// TwinCAT 3 PLC project EXERCISES
// ProgramVersion: 3.1.4023.0
// libraries:
//   CmpBitmapPool, * (System)
//   Tc2_Standard, * (Beckhoff Automation GmbH)
//   Tc2_System, * (Beckhoff Automation GmbH)
//   Tc2_Utilities, * (Beckhoff Automation GmbH)
//   Tc3_Module, * (Beckhoff Automation GmbH)
// project tree:
//   DUTs/ Pers_Data.TcDUT
//   / GlobalTextList.TcGTLO, ImagePool.TcIPO (not stored), PlcTask.TcTTO, Visualization Manager.TcVMO (not stored)
//   POUs/ Auto_Deur.TcPOU, Belsig_Winkeldeur.TcPOU, Check_Bounds_15_TO_24.TcPOU, FB_PULSE_PER_X_SEC.TcPOU, FB_PWM.TcPOU, Knipperlicht.TcPOU, MAIN.TcPOU, Open_Toilet.TcPOU, Parking.TcPOU, FC_SCALE.TcPOU, Product_Tellen_Verdelen.TcPOU, FB_String_Search.TcPOU, Trappenhuisautomaat.TcPOU
//   VISUs/ Auto_Deur.TcVIS, Belsig_Winkeldeur.TcVIS, Knipperlicht.TcVIS, Open_Toilet.TcVIS, Parking.TcVIS, Product_Tellen_Verdelen.TcVIS, Trappenhuisautomaat.TcVIS
// real-time tasks:
//   TASK PlcTask: cycle T#10ms, priority 20, ADS port 350

CONFIGURATION EXERCISES
    RESOURCE PLC ON TwinCAT3
        TASK PlcTask(INTERVAL := T#10ms, PRIORITY := 20);
        PROGRAM MAIN WITH PlcTask : MAIN;
    END_RESOURCE
END_CONFIGURATION

// ---- DUTs/Pers_Data.TcDUT
TYPE Pers_Data :
STRUCT
	Name : STRING;
	Firstname :  STRING;
	Age : STRING;
	Address : STRING;
END_STRUCT
END_TYPE

// ---- POUs/MAIN.TcPOU
PROGRAM MAIN
VAR
	KASPER : UINT;
	FB_PWM : FB_PWM;
	PWM : BOOL;
END_VAR

FB_PWM(DUTY:= 50, PERIOD_MS:= 4000);

PWM := FB_PWM.PWM_SIGNAL;

END_PROGRAM

// ---- POUs/FB_PWM.TcPOU
FUNCTION_BLOCK FB_PWM

VAR_INPUT
	DUTY : UINT;
	PERIOD_MS : UINT;
END_VAR

VAR_OUTPUT
	PWM_SIGNAL : BOOL;
END_VAR

VAR
	ON_TIME_STR : STRING;
	OFF_TIME_STR : STRING;
	
	ON_TIME : TIME;
	OFF_TIME : TIME;
	
	TON : TON;
	TOF : TOF;
END_VAR

ON_TIME_STR := UINT_TO_STRING(DUTY * PERIOD_MS / 100);
ON_TIME_STR := CONCAT('T#', ON_TIME_STR);
ON_TIME_STR := CONCAT(ON_TIME_STR, 'ms');
ON_TIME := STRING_TO_TIME(ON_TIME_STR);
	
OFF_TIME_STR := UINT_TO_STRING(PERIOD_MS - (DUTY * PERIOD_MS / 100));
OFF_TIME_STR := CONCAT('T#', OFF_TIME_STR);
OFF_TIME_STR := CONCAT(OFF_TIME_STR, 'ms');
OFF_TIME := STRING_TO_TIME(OFF_TIME_STR);

TOF(IN:= TON.Q, PT:= ON_TIME, Q => PWM_SIGNAL);
TON(IN:= NOT(TOF.Q), PT:= OFF_TIME);

END_FUNCTION_BLOCK

// ---- POUs/Auto_Deur.TcPOU
PROGRAM Auto_Deur
VAR
	TOF : TOF;
END_VAR

VAR_INPUT
	SW_MAIN : BOOL;
	SW_KASSA : BOOL;
	SENSOR_DOOR : BOOL;
END_VAR

VAR_OUTPUT
	CIL : BOOL;
END_VAR

IF SW_MAIN THEN
	TOF(IN:= SW_KASSA OR SENSOR_DOOR, PT:= T#1S, Q=> CIL);
END_IF

END_PROGRAM

// ---- POUs/Belsig_Winkeldeur.TcPOU
PROGRAM Belsig_Winkeldeur
VAR
	CTU : CTU;
	R_TRIG : R_TRIG;
	R_TRIG2 : R_TRIG;
END_VAR

VAR_INPUT
	S01 : BOOL;
	S02 : BOOL;
END_VAR

VAR_OUTPUT
	Q00 : BOOL;
END_VAR

CTU(CU := R_TRIG.Q);
R_TRIG(CLK := Q00);
R_TRIG2(CLK := S02);

IF S01 THEN
	IF R_TRIG2.Q THEN
		Q00 := TRUE;
	END_IF
	
ELSIF Q00 THEN
	IF S02 THEN
		Q00 := TRUE;
	ELSE
		Q00 := FALSE;
	END_IF
END_IF

END_PROGRAM

// ---- POUs/Check_Bounds_15_TO_24.TcPOU
FUNCTION Check_Bounds_15_TO_24 : BOOL

VAR_INPUT
	Value : UINT;
END_VAR

IF VALUE <= 24 AND VALUE >= 15 THEN
	Check_Bounds_15_TO_24 := TRUE;
ELSE
	Check_Bounds_15_TO_24 := FALSE;
END_IF

END_FUNCTION

// ---- POUs/FB_PULSE_PER_X_SEC.TcPOU
FUNCTION_BLOCK FB_PULSE_PER_X_SEC
VAR_INPUT
	ON_OFF : BOOL;
	X_Sec : UINT;
END_VAR

VAR_OUTPUT
	PULSE : BOOL;
END_VAR

VAR
	R_TRIG : R_TRIG;
	TIMETIME : TIME;
	TIME_TIJD : STRING;
	TON : TON;
	TOF : TOF;
END_VAR

TIME_TIJD := CONCAT('T#', UINT_TO_STRING(X_Sec));
TIME_TIJD := CONCAT(TIME_TIJD, 's');

TOF(IN:= TON.Q, PT:= T#0MS);
TON(IN:= NOT(TOF.Q), PT:= STRING_TO_TIME(TIME_TIJD), Q => Pulse);

END_FUNCTION_BLOCK

// ---- POUs/Knipperlicht.TcPOU
PROGRAM Knipperlicht
VAR
	TOF : TOF;
	TON : TON;
END_VAR

VAR_OUTPUT
	LAMP : BOOL;
END_VAR

TOF(IN:= TON.Q, PT:= T#500MS, Q => LAMP);
TON(IN:= NOT(TOF.Q), PT:= T#500ms);

END_PROGRAM

// ---- POUs/Open_Toilet.TcPOU
PROGRAM Open_Toilet
VAR
	TOF : TOF;
END_VAR

VAR_INPUT
	SW1 : BOOL; // SWITCH 1
	SW2 : BOOL; // SWITCH 2
	SW3 : BOOL; // SWITCH 3
END_VAR

VAR_OUTPUT
	Q00 : BOOL; // VENTILATOR
	Q01 : BOOL; // LAMP 1
	Q02 : BOOL; // LAMP 2
	Q03 : BOOL; // LAMP 3
END_VAR

TOF(IN:= SW1 OR SW2 OR SW3, PT:= T#5S, Q=> Q00);

END_PROGRAM

// ---- POUs/Parking.TcPOU
PROGRAM Parking
VAR
	R_TRIG_1 : R_TRIG;
	R_TRIG_2 : R_TRIG;
	
	R_TRIG_BINNEN : R_TRIG;
	R_TRIG_BUITEN : R_TRIG;
	
	CTUD : CTUD;	
	
	PING1 : BOOL;
	PING2 : BOOL;
	
	BINNEN : BOOL;
	BUITEN : BOOL;
END_VAR

VAR_INPUT
	SENSOR_1 : BOOL;
	SENSOR_2 : BOOL;
END_VAR

VAR_OUTPUT
	LED_R : BOOL;
	LED_G : BOOL;
	SLAGBOOM : BOOL;
END_VAR

R_TRIG_1(CLK := SENSOR_1);
R_TRIG_2(CLK := SENSOR_2);
R_TRIG_BINNEN(CLK := BINNEN);
R_TRIG_BUITEN(CLK := BUITEN);

CTUD(CU := R_TRIG_BINNEN.Q, CD := R_TRIG_BUITEN.Q);

IF R_TRIG_1.Q THEN
	IF PING2 THEN
		BUITEN := TRUE;
		SLAGBOOM := FALSE;
		PING2 := FALSE;
	ELSE
		PING1 := TRUE;
		SLAGBOOM := TRUE;
	END_IF
ELSE
	BUITEN := FALSE;
END_IF

IF R_TRIG_2.Q THEN
	IF PING1 THEN
		BINNEN := TRUE;
		SLAGBOOM := FALSE;
		PING1 := FALSE;
	ELSE
		PING2 := TRUE;
		SLAGBOOM := TRUE;
	END_IF
ELSE
	BINNEN := FALSE;
END_IF

IF CTUD.CV < 10 THEN
	LED_G := TRUE;
	LED_R := FALSE;
ELSE
	LED_R := TRUE;
	LED_G := FALSE;
END_IF

END_PROGRAM

// ---- POUs/FC_SCALE.TcPOU
FUNCTION FC_SCALE : LREAL

VAR_INPUT
	RawValue : LREAL;
	Rvmin : LREAL;
	Rvmax : LREAL;
	SVmin : LREAL;
	SVmax : LREAL;
END_VAR

FC_SCALE := SVmin + (RawValue / ((Rvmax-Rvmin)/(SVmax-SVmin)));

END_FUNCTION

// ---- POUs/Product_Tellen_Verdelen.TcPOU
PROGRAM Product_Tellen_Verdelen
VAR
	R_TRIG : R_TRIG;
	CTU : CTU;
END_VAR

VAR_INPUT
	SENSOR : BOOL;
	STAND_1 : BOOL;
	STAND_2 : BOOL;
END_VAR

VAR_OUTPUT
END_VAR

R_TRIG(CLK := SENSOR);
CTU(CU:= R_TRIG.Q); 

IF CTU.CV < 10 THEN
	CTU.RESET := FALSE;
	STAND_1 := TRUE;
	STAND_2 := FALSE;
ELSIF CTU.CV < 30 THEN
	STAND_1 := FALSE;
	STAND_2 := TRUE;
ELSE
	CTU.RESET := R_TRIG.Q;
END_IF

END_PROGRAM

// ---- POUs/FB_String_Search.TcPOU
FUNCTION_BLOCK FB_String_Search

VAR_INPUT
	InputString : Pers_Data;
	SearchString : STRING;
END_VAR

VAR_OUTPUT
	OUT : BOOL;
END_VAR

VAR
	SUB_STRING : STRING;
END_VAR

SUB_STRING := CONCAT(SUB_STRING, InputString.Name);
SUB_STRING := CONCAT(SUB_STRING, InputString.Firstname);
SUB_STRING := CONCAT(SUB_STRING, InputString.Age);
SUB_STRING := CONCAT(SUB_STRING, InputString.Address);

OUT := INT_TO_BOOL(FIND(STR1:= F_ToLCase(SUB_String), STR2:= F_ToLCase(SearchString)));

END_FUNCTION_BLOCK

// ---- POUs/Trappenhuisautomaat.TcPOU
PROGRAM Trappenhuisautomaat
VAR
	TOF : TOF;
	CTUD : CTUD;
END_VAR

VAR_INPUT
	SW0 : BOOL;
	SW1 : BOOL;
	SW2 : BOOL;
	SW3 : BOOL;
	SW4 : BOOL;
	SW5 : BOOL;
	SW6 : BOOL;
END_VAR

VAR_OUTPUT
	Q01 : BOOL;
END_VAR

TOF(IN:= SW0, PT:= T#3S, Q=> Q01);
CTUD.RESET := NOT(Q01);


IF SW1 OR SW2 OR SW3 OR SW4 OR SW5 OR SW6 THEN
	SW0 := TRUE; 
	CTUD.CU := SW0;
	IF CTUD.CV = 2 THEN
		TOF.PT := T#0S;
		SW0 := FALSE;
		Q01 := FALSE; 
	END_IF
ELSE
	SW0 := FALSE;
END_IF

END_PROGRAM

// ---- GlobalTextList.TcGTLO
TEXTLIST GlobalTextList
  868 = '%d'
  584 = '%ld'
END_TEXTLIST

// ---- VISUs/Auto_Deur.TcVIS
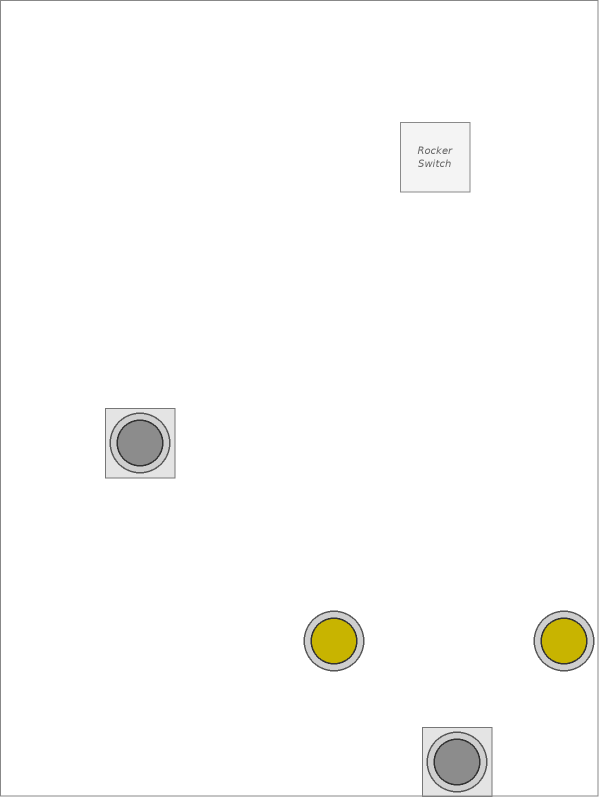
VISUALIZATION Auto_Deur  // 599x797
    Lamp1 (529,606 70x70), variable: Auto_Deur.CIL, style: Lamp-Lamp1-Yellow
    Lamp1 (299,606 70x70), variable: Auto_Deur.CIL, style: Lamp-Lamp1-Yellow
    PushSwitch (422,727 70x70), variable: Auto_Deur.SENSOR_DOOR, behaviour: TAP, style: Switch-PushSwitch-Gray
    PushSwitch (105,408 70x70), variable: Auto_Deur.SW_KASSA, behaviour: TAP, style: Switch-PushSwitch-Gray
    RockerSwitch (400,122 70x70), variable: Auto_Deur.SW_MAIN, behaviour: TOGGLE, style: Switch-RockerSwitch-Gray
END_VISUALIZATION

// ---- VISUs/Belsig_Winkeldeur.TcVIS
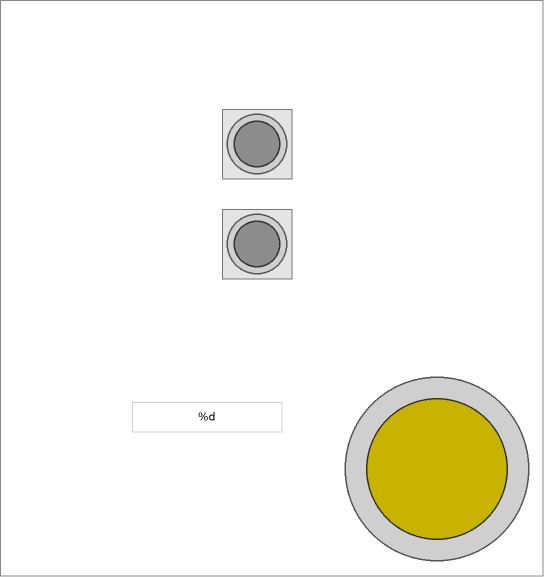
VISUALIZATION Belsig_Winkeldeur  // 544x577
    PushSwitch (222,109 70x70), variable: Belsig_Winkeldeur.S01, behaviour: TOGGLE, style: Switch-PushSwitch-Gray
    PushSwitch (222,209 70x70), variable: Belsig_Winkeldeur.S02, behaviour: TOGGLE, style: Switch-PushSwitch-Gray
    Lamp1 (330,361 214x216), variable: Belsig_Winkeldeur.Q00, style: Lamp-Lamp1-Yellow
    Textfield (132,402 150x30), "%d", text variable: Belsig_Winkeldeur.CTU.CV
END_VISUALIZATION

// ---- VISUs/Knipperlicht.TcVIS
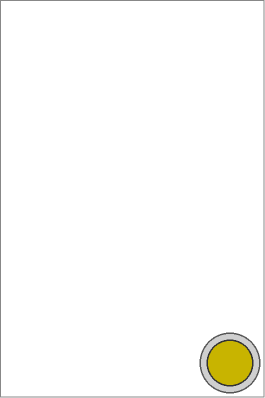
VISUALIZATION Knipperlicht  // 265x398
    Lamp1 (195,328 70x70), variable: Knipperlicht.LAMP, style: Lamp-Lamp1-Yellow
END_VISUALIZATION

// ---- VISUs/Open_Toilet.TcVIS
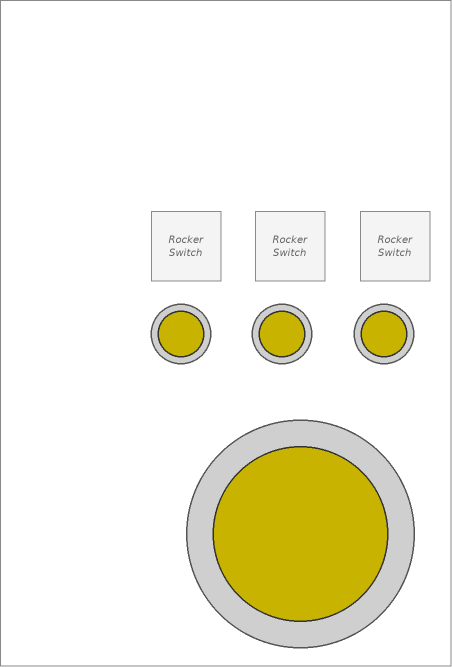
VISUALIZATION Open_Toilet  // 452x667
    Lamp1 (146,299 70x70), variable: Open_Toilet.SW1, style: Lamp-Lamp1-Yellow
    Lamp1 (247,299 70x70), variable: Open_Toilet.SW2, style: Lamp-Lamp1-Yellow
    Lamp1 (349,299 70x70), variable: Open_Toilet.SW3, style: Lamp-Lamp1-Yellow
    Lamp1 (149,401 303x266), variable: Open_Toilet.Q00, style: Lamp-Lamp1-Yellow
    RockerSwitch (151,211 70x70), variable: Open_Toilet.SW1, behaviour: TOGGLE, style: Switch-RockerSwitch-Gray
    RockerSwitch (255,211 70x70), variable: Open_Toilet.SW2, behaviour: TOGGLE, style: Switch-RockerSwitch-Gray
    RockerSwitch (360,211 70x70), variable: Open_Toilet.SW3, behaviour: TOGGLE, style: Switch-RockerSwitch-Gray
END_VISUALIZATION

// ---- VISUs/Parking.TcVIS
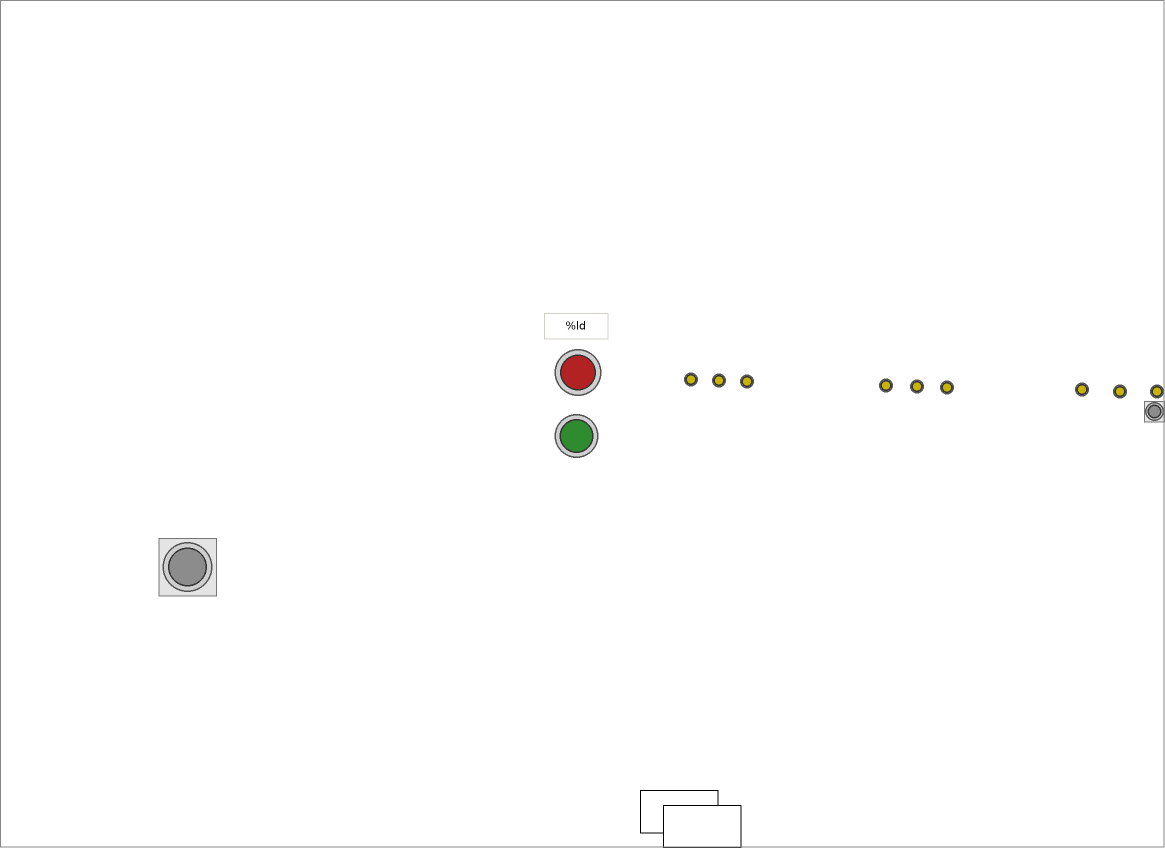
VISUALIZATION Parking  // 1165x848, background image ImagePool.image-3
    Lamp1 (551,345 54x55), variable: Parking.LED_R, style: Lamp-Lamp1-Red
    Lamp1 (551,410 51x52), variable: Parking.LED_G, style: Lamp-Lamp1-Green
    Textfield (544,313 64x26), "%ld", text variable: Parking.CTUD.CV
    PushSwitch (1144,399 21x25), variable: Parking.SENSOR_2, behaviour: TAP, style: Switch-PushSwitch-Gray
    PushSwitch (158,538 59x58), variable: Parking.SENSOR_1, behaviour: TAP, style: Switch-PushSwitch-Gray
    Rectangle (640,790 78x43), angle 69
    Rectangle (663,805 78x43), angle 160
    Lamp1 (683,359 16x41), variable: Parking.SLAGBOOM, style: Lamp-Lamp1-Yellow
    Lamp1 (711,360 16x41), variable: Parking.SLAGBOOM, style: Lamp-Lamp1-Yellow
    Lamp1 (739,361 16x41), variable: Parking.SLAGBOOM, style: Lamp-Lamp1-Yellow
    Lamp1 (878,365 16x41), variable: Parking.SLAGBOOM, style: Lamp-Lamp1-Yellow
    Lamp1 (939,367 16x41), variable: Parking.SLAGBOOM, style: Lamp-Lamp1-Yellow
    Lamp1 (909,366 16x41), variable: Parking.SLAGBOOM, style: Lamp-Lamp1-Yellow
    Lamp1 (1074,369 16x41), variable: Parking.SLAGBOOM, style: Lamp-Lamp1-Yellow
    Lamp1 (1112,370 16x43), variable: Parking.SLAGBOOM, style: Lamp-Lamp1-Yellow
    Lamp1 (1149,371 16x41), variable: Parking.SLAGBOOM, style: Lamp-Lamp1-Yellow
END_VISUALIZATION

// ---- VISUs/Product_Tellen_Verdelen.TcVIS
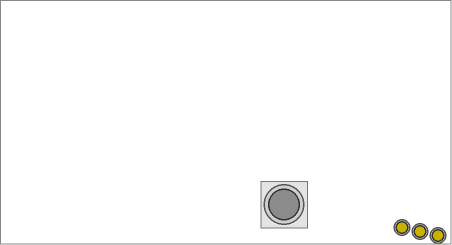
VISUALIZATION Product_Tellen_Verdelen  // 452x245, background image ImagePool.VerdelerFULL
    PushSwitch (259,181 50x47), variable: Product_Tellen_Verdelen.SENSOR, behaviour: TAP, style: Switch-PushSwitch-Gray
    Lamp1 (388,218 28x19), variable: Product_Tellen_Verdelen.STAND_2, style: Lamp-Lamp1-Yellow
    Lamp1 (406,222 28x19), variable: Product_Tellen_Verdelen.STAND_2, style: Lamp-Lamp1-Yellow
    Lamp1 (424,226 28x19), variable: Product_Tellen_Verdelen.STAND_2, style: Lamp-Lamp1-Yellow
END_VISUALIZATION

// ---- VISUs/Trappenhuisautomaat.TcVIS
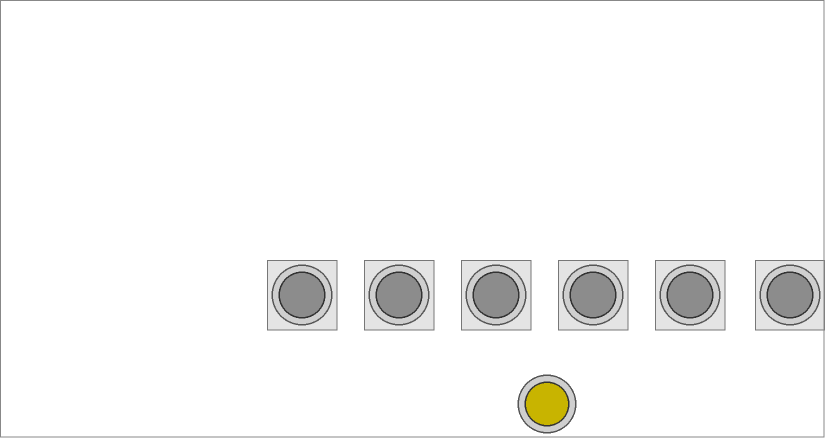
VISUALIZATION Trappenhuisautomaat  // 825x438
    Lamp1 (512,370 70x68), variable: Trappenhuisautomaat.Q01, style: Lamp-Lamp1-Yellow
    PushSwitch (267,260 70x70), variable: Trappenhuisautomaat.SW1, behaviour: TAP, style: Switch-PushSwitch-Gray
    PushSwitch (755,260 70x70), variable: Trappenhuisautomaat.SW6, behaviour: TAP, style: Switch-PushSwitch-Gray
    PushSwitch (655,260 70x70), variable: Trappenhuisautomaat.SW5, behaviour: TAP, style: Switch-PushSwitch-Gray
    PushSwitch (558,260 70x70), variable: Trappenhuisautomaat.SW4, behaviour: TAP, style: Switch-PushSwitch-Gray
    PushSwitch (364,260 70x70), variable: Trappenhuisautomaat.SW2, behaviour: TAP, style: Switch-PushSwitch-Gray
    PushSwitch (461,260 70x70), variable: Trappenhuisautomaat.SW3, behaviour: TAP, style: Switch-PushSwitch-Gray
END_VISUALIZATION
